(* CoDeSys 2.3.9.50 project: 8B.pr6 *)
(* Libraries: STANDARD.LB6 5.6.98 12:03:02 *)

(* POU MAIN, LD *)
PROGRAM MAIN
VAR
	Start AT %IX0.0: BOOL;
	Conveyer_Start AT %QX0.0: BOOL;
	Stop AT %IX0.1: BOOL;
	Temp_Stop AT %QX0.1: BOOL;
	Running AT %QX0.2: BOOL;
	Stand_By AT %QX0.3: BOOL;
	Box_Sensed AT %IX0.2: BOOL;
	Photo_Sensor AT %QX0.4: BOOL;
	Solenoid AT %QX0.5: BOOL;
	Filling_Start AT %QX0.6: BOOL;
	Box_Full AT %IX0.3: BOOL;
	Box_Sensed_Full AT %QX0.7: BOOL;
	Full_light AT %QX1.0: BOOL;
END_VAR
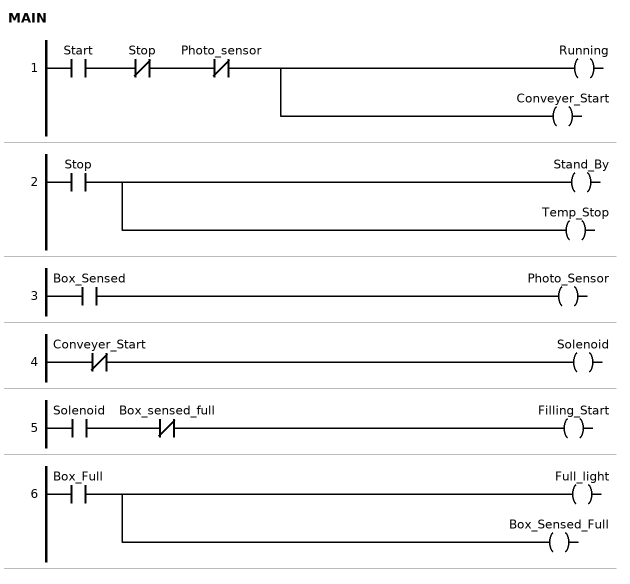
_LD_ (* Ladder Diagram *)
NETWORK 1
	[Start] - [/Stop] - [/Photo_sensor] --- (Running) (Conveyer_Start)
NETWORK 2
	[Stop] --- (Stand_By) (Temp_Stop)
NETWORK 3
	[Box_Sensed] --- (Photo_Sensor)
NETWORK 4
	[/Conveyer_Start] --- (Solenoid)
NETWORK 5
	[Solenoid] - [/Box_sensed_full] --- (Filling_Start)
NETWORK 6
	[Box_Full] --- (Full_light) (Box_Sensed_Full)
_END_LD_
(* the same logic as Structured Text *)
(* Network 1 *)
Running := Start AND NOT Stop AND NOT Photo_sensor;
Conveyer_Start := Running;
(* Network 2 *)
Stand_By := Stop;
Temp_Stop := Stop;
(* Network 3 *)
Photo_Sensor := Box_Sensed;
(* Network 4 *)
Solenoid := NOT Conveyer_Start;
(* Network 5 *)
Filling_Start := Solenoid AND NOT Box_sensed_full;
(* Network 6 *)
Full_light := Box_Full;
Box_Sensed_Full := Box_Full;
END_PROGRAM
